INTERFACE I_ListNode EXTENDS I_CollectionNode;

END_INTERFACE

(* stored: Version 1.1.0.1, ProductVersion 3.1.4024.12
   Itf I_ListNode: Id {052a77a7-47a6-4fd1-a8c8-be2a68400d3d} *)
